// TIA Portal V20 export
FUNCTION "EM8_TeachingData" : Void   // FC86, LAD
// stored: Namespace Unit1.Em8, SetENOAutomatically false
BEGIN

REGION Network 2 (SCL): Thickness AxisZ Teaching Data
   //Thickness AxisZ Position 0
   "Unit1.Em8.HmiInterface".cmThicknessAxisZ.configuration.setPositions[0].position := 0.0;
   "Unit1.Em8.HmiInterface".cmThicknessAxisZ.configuration.setPositions[0].velocity := 30.0;
   "Unit1.Em8.HmiInterface".cmThicknessAxisZ.configuration.setPositions[0].acceleration := 300.0;
   "Unit1.Em8.HmiInterface".cmThicknessAxisZ.configuration.setPositions[0].deceleration := 300.0;

   //Thickness AxisZ Position 1
   "Unit1.Em8.HmiInterface".cmThicknessAxisZ.configuration.setPositions[1].position := 80.0;
   "Unit1.Em8.HmiInterface".cmThicknessAxisZ.configuration.setPositions[1].velocity := 30.0;
   "Unit1.Em8.HmiInterface".cmThicknessAxisZ.configuration.setPositions[1].acceleration := 300.0;
   "Unit1.Em8.HmiInterface".cmThicknessAxisZ.configuration.setPositions[1].deceleration := 300.0;

   //Thickness AxisZ Position 2
   "Unit1.Em8.HmiInterface".cmThicknessAxisZ.configuration.setPositions[2].position := 90.0;
   "Unit1.Em8.HmiInterface".cmThicknessAxisZ.configuration.setPositions[2].velocity := 10.0;
   "Unit1.Em8.HmiInterface".cmThicknessAxisZ.configuration.setPositions[2].acceleration := 100.0;
   "Unit1.Em8.HmiInterface".cmThicknessAxisZ.configuration.setPositions[2].deceleration := 100.0;
END_REGION
END_FUNCTION
